// TIA Portal V18 export
// export: Created 2025-12-01T17:51:17.873891Z, ExportSetting None, DisplayName Totally Integrated Automation Portal, DisplayVersion V18 Update 5, DisplayName TIA Portal Openness, DisplayVersion V18 Update 5, DisplayName TIA Portal Teamcenter Gateway, DisplayVersion V18, DisplayName TIA Portal Version Control Interface, DisplayVersion V18, DisplayName STEP 7 Professional, DisplayVersion V18 Update 5, DisplayName STEP 7 Safety, DisplayVersion V18, DisplayName WinCC Professional, DisplayVersion V18 Update 5
DATA_BLOCK "ServoV90_A3"   // DB2503
{ S7_Optimized_Access := 'FALSE' }
// stored: AutoNumber false
   VAR
      In : Struct
         iInterlock : Bool := TRUE;   // interlock
         "iManJog+" : Bool := FALSE;   // positive motion/action/...manually
         "iManJog-" : Bool := FALSE;   // negtive motion/action/...manually
         iAutoStart : Bool := FALSE;   // negtive motion/action/...automaticly
         iHome : Bool := FALSE;   // Homing
         iCancelTask : Bool := FALSE;   // Cancel task
         iPauseTask : Bool := FALSE;   // Pause task
         iManStart : Bool := FALSE;   // positive motion/action/...automaticly
         iManListStart : Bool := FALSE;
         iLimitSwitchActive : Bool := TRUE;
         iLimitSoftActive : Bool := TRUE;
         iRunningTimeout : Time := T#0MS;
         iHomingTimeout : Time := T#0MS;
         iAutoPosition : DInt := 0;
         iAutoVelocity : Int := 0;
         iManListPosition : DInt := 0;
         iManListVelocity : Int := 0;
         iManListNumber : Int := 0;   // position list number
         iManPosition : DInt := 0;
         iManVelocity : Int := 0;
         iMode : Int := 0;   // 1-相对;2-绝对
      END_STRUCT;
      Out : Struct
         oReady : Bool := FALSE;
         oWarning : Bool := FALSE;   // warning
         oError : Bool := TRUE;   // error
         oInterlock : Bool := TRUE;
         oServoEnable : Bool := FALSE;
         oRunning : Bool := FALSE;
         oHoming : Bool := FALSE;
         oHomeRef : Bool := TRUE;
         oServoPosOK : Bool := FALSE;
         oErrorCode : Int := -244;
         oStatus : Int := 0;
         oActPosition : DInt := -3;
         oManualListPos : DInt := 0;
      END_STRUCT;
      IO : Struct
         ioManEnale : Bool := FALSE;
         ioAutoEnale : Bool := FALSE;
         ioAutoHome : Bool;
      END_STRUCT;
      Spare : Struct
         S : Array[0..100] of Byte;
      END_STRUCT;
      Manual : Struct
         Index : Int := 1;
         Pos : Array[1..20] of Struct
            Pos : DInt;
            Vel : Int;
         END_STRUCT;
      END_STRUCT;
      Auto : Struct
         Index : Int := 1;
         Pos : Array[1..20] of Struct
            Pos : DInt;
            Vel : Int;
         END_STRUCT;
      END_STRUCT;
      Interlock : Struct
         Active : Bool := FALSE;
         Case1 : Bool := TRUE;
         Case2 : Bool := TRUE;
         Case3 : Bool := FALSE;
         Case4 : Bool := FALSE;
         Case5 : Bool := FALSE;
         Case6 : Bool := FALSE;
         Case7 : Bool := FALSE;
         Case8 : Bool := FALSE;
         Case9 : Bool := FALSE;
         Case10 : Bool := FALSE;
      END_STRUCT;
      PositionOk : Array[1..20] of Bool;
      Home_Pos : Struct
         "Home Pos Pls" : Bool := FALSE;
         "Arrow indication" : Int := 0;
         "Process prompt" : Int := 0;
         "Button prompt" : Int := 0;
      END_STRUCT;
   END_VAR
BEGIN
   Spare.S[0..100] := 16#00;
   Manual.Pos[1].Pos := 0;
   Manual.Pos[2..6].Pos := 680000;
   Manual.Pos[7].Pos := 90000;
   Manual.Pos[8].Pos := 180000;
   Manual.Pos[9].Pos := 270000;
   Manual.Pos[10..20].Pos := 0;
   Manual.Pos[1].Vel := 20000;
   Manual.Pos[2..9].Vel := 10000;
   Manual.Pos[10..20].Vel := 0;
   Auto.Pos[1].Pos := 0;
   Auto.Pos[2..6].Pos := 680000;
   Auto.Pos[7].Pos := 90000;
   Auto.Pos[8].Pos := 180000;
   Auto.Pos[9].Pos := 270000;
   Auto.Pos[10..20].Pos := 0;
   Auto.Pos[1].Vel := 20000;
   Auto.Pos[2..9].Vel := 10000;
   Auto.Pos[10..20].Vel := 0;
   // Auto.Pos[1] : 1.取料位置
   // Auto.Pos[2] : 2.放料位置
   // Auto.Pos[3] : 3.
   // Auto.Pos[4] : 4.
   // Auto.Pos[5] : 5.
   // Auto.Pos[6] : 6.
   // Auto.Pos[7] : 7.
   // Auto.Pos[8] : 8.
   // Auto.Pos[9] : 9.
   PositionOk[1] := FALSE;   // [1]
   PositionOk[2] := FALSE;   // [2]
   PositionOk[3] := FALSE;   // [3]
   PositionOk[4] := FALSE;   // [4]
   PositionOk[5] := FALSE;   // [5]
   PositionOk[6] := FALSE;   // [6]
   PositionOk[7] := FALSE;   // [7]
   PositionOk[8] := FALSE;   // [8]
   PositionOk[9] := FALSE;   // [9]
   PositionOk[10..20] := FALSE;
END_DATA_BLOCK
